% RSLogix 500 project PV4.RSS, saved by version 8.30.00.16 %
PROJECT "PV4"    % processor: Bul.1763 MicroLogix 1100 Series B %

PROGRAM FILES
  LAD 2   20 rungs

DATA FILES
  O0 OUTPUT  5 elements
  I1 INPUT  7 elements
  S2 STATUS  66 elements
  B3 BINARY  2 elements
  T4 TIMER  2 elements
  C5 COUNTER  1 elements
  R6 CONTROL  1 elements
  N7 INTEGER  3 elements
  F8 FLOAT  1 elements

LADDER 2
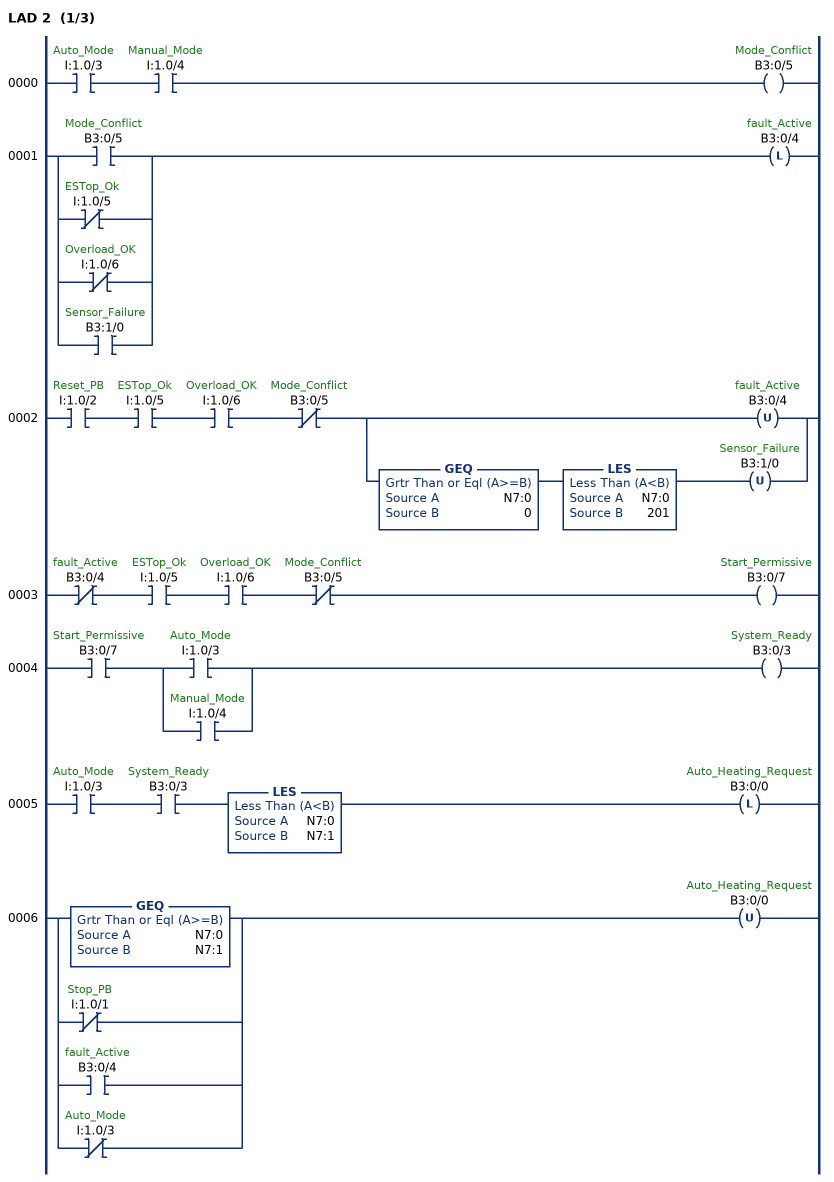
% Rung: 0 %
SOR XIC I:1.0/3 XIC I:1.0/4 OTE B3:0/5 EOR
%   I:1.0/3  "Auto_Mode" %
%   I:1.0/4  "Manual_Mode" %
%   B3:0/5  "Mode_Conflict" %
% Rung: 1 %
SOR BST XIC B3:0/5 NXB BST XIO I:1.0/5 NXB BST XIO I:1.0/6 NXB XIC B3:1/0 BND BND BND OTL B3:0/4 EOR
%   B3:0/5  "Mode_Conflict" %
%   I:1.0/5  "ESTop_Ok" %
%   I:1.0/6  "Overload_OK" %
%   B3:1/0  "Sensor_Failure" %
%   B3:0/4  "fault_Active" %
% Rung: 2 %
SOR XIC I:1.0/2 XIC I:1.0/5 XIC I:1.0/6 XIO B3:0/5 BST OTU B3:0/4 NXB GEQ N7:0 0 LES N7:0 201 OTU B3:1/0 BND EOR
%   I:1.0/2  "Reset_PB" %
%   I:1.0/5  "ESTop_Ok" %
%   I:1.0/6  "Overload_OK" %
%   B3:0/5  "Mode_Conflict" %
%   B3:0/4  "fault_Active" %
%   B3:1/0  "Sensor_Failure" %
% Rung: 3 %
SOR XIO B3:0/4 XIC I:1.0/5 XIC I:1.0/6 XIO B3:0/5 OTE B3:0/7 EOR
%   B3:0/4  "fault_Active" %
%   I:1.0/5  "ESTop_Ok" %
%   I:1.0/6  "Overload_OK" %
%   B3:0/5  "Mode_Conflict" %
%   B3:0/7  "Start_Permissive" %
% Rung: 4 %
SOR XIC B3:0/7 BST XIC I:1.0/3 NXB XIC I:1.0/4 BND OTE B3:0/3 EOR
%   B3:0/7  "Start_Permissive" %
%   I:1.0/3  "Auto_Mode" %
%   I:1.0/4  "Manual_Mode" %
%   B3:0/3  "System_Ready" %
% Rung: 5 %
SOR XIC I:1.0/3 XIC B3:0/3 LES N7:0 N7:1 OTL B3:0/0 EOR
%   I:1.0/3  "Auto_Mode" %
%   B3:0/3  "System_Ready" %
%   B3:0/0  "Auto_Heating_Request" %
% Rung: 6 %
SOR BST GEQ N7:0 N7:1 NXB BST XIO I:1.0/1 NXB BST XIC B3:0/4 NXB XIO I:1.0/3 BND BND BND OTU B3:0/0 EOR
%   I:1.0/1  "Stop_PB" %
%   B3:0/4  "fault_Active" %
%   I:1.0/3  "Auto_Mode" %
%   B3:0/0  "Auto_Heating_Request" %

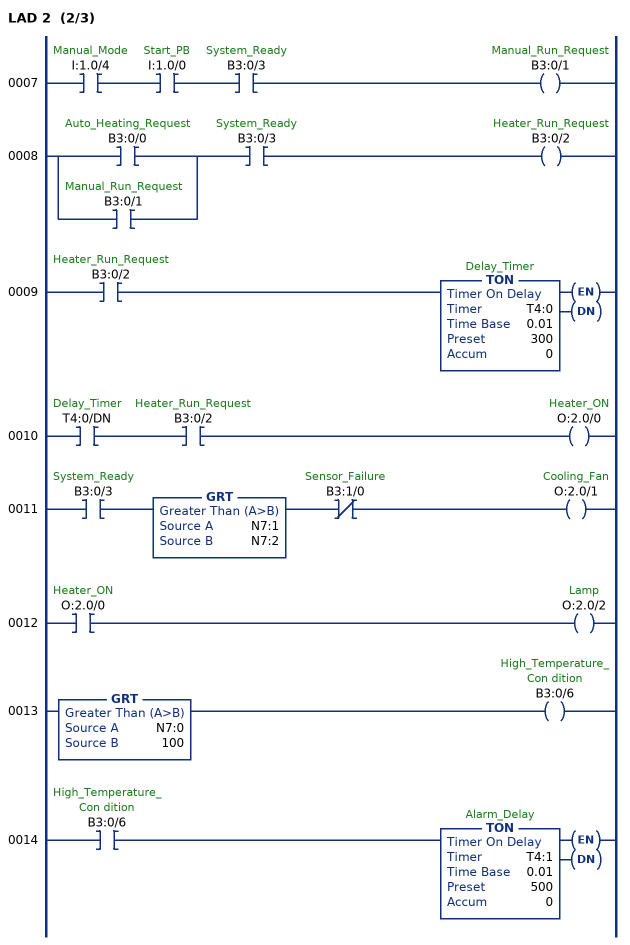
% Rung: 7 %
SOR XIC I:1.0/4 XIC I:1.0/0 XIC B3:0/3 OTE B3:0/1 EOR
%   I:1.0/4  "Manual_Mode" %
%   I:1.0/0  "Start_PB" %
%   B3:0/3  "System_Ready" %
%   B3:0/1  "Manual_Run_Request" %
% Rung: 8 %
SOR BST XIC B3:0/0 NXB XIC B3:0/1 BND XIC B3:0/3 OTE B3:0/2 EOR
%   B3:0/0  "Auto_Heating_Request" %
%   B3:0/1  "Manual_Run_Request" %
%   B3:0/3  "System_Ready" %
%   B3:0/2  "Heater_Run_Request" %
% Rung: 9 %
SOR XIC B3:0/2 TON T4:0 0.01 300 0 EOR
%   B3:0/2  "Heater_Run_Request" %
%   T4:0  "Delay_Timer" %
% Rung: 10 %
SOR XIC T4:0/DN XIC B3:0/2 OTE O:2.0/0 EOR
%   T4:0  "Delay_Timer" %
%   B3:0/2  "Heater_Run_Request" %
%   O:2.0/0  "Heater_ON" %
% Rung: 11 %
SOR XIC B3:0/3 GRT N7:1 N7:2 XIO B3:1/0 OTE O:2.0/1 EOR
%   B3:0/3  "System_Ready" %
%   B3:1/0  "Sensor_Failure" %
%   O:2.0/1  "Cooling_Fan" %
% Rung: 12 %
SOR XIC O:2.0/0 OTE O:2.0/2 EOR
%   O:2.0/0  "Heater_ON" %
%   O:2.0/2  "Lamp" %
% Rung: 13 %
SOR GRT N7:0 100 OTE B3:0/6 EOR
%   B3:0/6  "High_Temperature_Con dition" %
% Rung: 14 %
SOR XIC B3:0/6 TON T4:1 0.01 500 0 EOR
%   B3:0/6  "High_Temperature_Con dition" %
%   T4:1  "Alarm_Delay" %

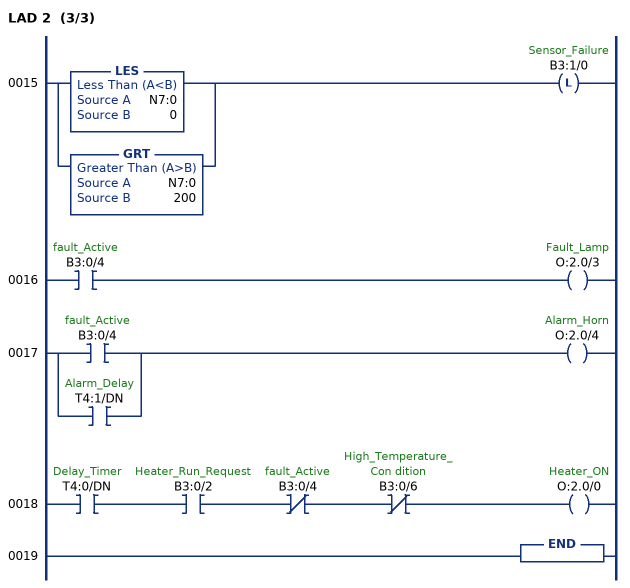
% Rung: 15 %
SOR BST LES N7:0 0 NXB GRT N7:0 200 BND OTL B3:1/0 EOR
%   B3:1/0  "Sensor_Failure" %
% Rung: 16 %
SOR XIC B3:0/4 OTE O:2.0/3 EOR
%   B3:0/4  "fault_Active" %
%   O:2.0/3  "Fault_Lamp" %
% Rung: 17 %
SOR BST XIC B3:0/4 NXB XIC T4:1/DN BND OTE O:2.0/4 EOR
%   B3:0/4  "fault_Active" %
%   T4:1  "Alarm_Delay" %
%   O:2.0/4  "Alarm_Horn" %
% Rung: 18 %
SOR XIC T4:0/DN XIC B3:0/2 XIO B3:0/4 XIO B3:0/6 OTE O:2.0/0 EOR
%   T4:0  "Delay_Timer" %
%   B3:0/2  "Heater_Run_Request" %
%   B3:0/4  "fault_Active" %
%   B3:0/6  "High_Temperature_Con dition" %
%   O:2.0/0  "Heater_ON" %
% Rung: 19 %
SOR END EOR

OTHER DOCUMENTED ADDRESSES
  I:1.0/7  "Low_Level_Switch"
  I:1.0/8  "High_Level_Switch"
  I:3.0/0  "High_Level_Switch"
  O:2.0/5  "High_Level_Lamp"

DATA TABLE (non-zero values as saved)
DATA B3
% B3:0 % 0X0088 0X0000
DATA T4
% .PRE .ACC %
% T4:0 % 300 0
% T4:1 % 500 0
DATA N7
% N7:0 % 70 70 75
